FUNCTION_BLOCK ConexionEthernet IMPLEMENTS I_Conexion

VAR
//    rtMessageOutput: R_TRIG; (* Declaration *)
//    bFeedTooHigh: BOOL;
    udiAdsLogRes: UDINT;
END_VAR


METHOD EstablecerConexion : BOOL
//rtMessageOutput(CLK := bFeedTooHigh);
//IF rtMessageOutput.Q THEN 
    UdiAdsLogRes := ADSLOGDINT( msgCtrlMask := ADSLOG_MSGTYPE_HINT OR ADSLOG_MSGTYPE_MSGBOX, 
                    msgFmtStr := 'PLC Mensaje: estamos realizando una conexión por Ethernet: %d', dintArg:= 1);
//END_IF
END_METHOD

END_FUNCTION_BLOCK

(* stored: Version 1.1.0.1, ProductVersion 3.1.4024.12
   POU ConexionEthernet: Id {f1b3daed-ef99-475d-a42a-a1fa58efccc1}, SpecialFunc None
   Method EstablecerConexion: Id {30ebfe30-4904-4613-8b60-ac39ab4d8fff} *)
